FUNCTION_BLOCK AlPgnRxNew8Bcylc_REQ (* Service Interface Function Block Type *)
  (* Standard: 61499-2 *)
  (* Version 1.0, 2025-09-04, franz *)
  PACKAGE isobus::rx;
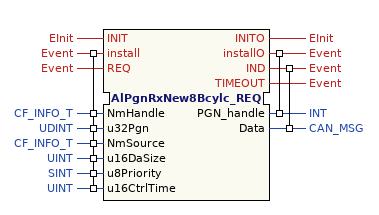
  EVENT_INPUT
    INIT : EInit; (* Service Initialization *)
    install WITH NmHandle, u32Pgn, NmSource, u16DaSize, u8Priority, u16CtrlTime; (* installs a Transmit PGN (TX) *)
    REQ; (* This function releases the cyclic sending of requests for a RX PGN *)
  END_EVENT
  EVENT_OUTPUT
    INITO : EInit; (* Initialization Confirm *)
    installO WITH PGN_handle; (* install Done *)
    IND WITH Data; (* Data was received *)
    TIMEOUT;
  END_EVENT
  VAR_INPUT
    NmHandle : isobus::CF_INFO_T; (* Handle of network member assigned of Network management *)
    u32Pgn : UDINT; (* PGN - Range: 0 - 0x3FFFF *)
    NmSource : isobus::CF_INFO_T; (* Define the Communication Partner *)
    u16DaSize : UINT; (* Data length of this PGN (0..8) *)
    u8Priority : SINT; (* Default priority of this PGN (0..7) 0=highest *)
    u16CtrlTime : UINT; (* 0 ... 0xFDFF ms *)
  END_VAR
  VAR_OUTPUT
    PGN_handle : INT; (* PGN-handle on success, HANDLE_UNVALID in case of an error *)
    Data : isobus::CAN_MSG;
  END_VAR
END_FUNCTION_BLOCK
